{attribute 'GeneratedUsingTerminal: EP1312-0001-0016'}
{attribute addProperty BoxType "EP1312-0001-0016"}
{attribute addProperty Id "A_0038_EP1518_0002_0016EP1518_CC44258859A_0039_EP1518_0002_0017EP1518_CC44258859A_0040_EP1518_0002_0018EP1518_CC44258859A_0041_EP1518_0002_0019EP1518_CC44258859A_0042_EP1809_0021_0016EP1809_32157CFD20A_0043_EP1809_0021_0017EP1809_32157CFD20A_0044_EP1809_0022_0017EP1809_32157CFD20A_0045_EP1809_0022_0018EP1809_32157CFD20A_0046_EP1809_0042_0018EP1809_AA84A50E20A_0047_EP1809_0042_0019EP1809_8E14C81620A_0048_EP1816_0003_0016EP1816_73178B5432A_0049_EP1816_0008_0016EP1816_03D8810930A_0050_EP1816_0008_0017EP1816_03D8810930A_0051_EP1816_0008_0018EP1816_5E50D3DD30A_0052_EP1816_0008_0019EP1816_5E50D3DD30A_0053_EP1816_0008_0020EP1816_5E50D3DD30A_0054_EP1816_1008_0016EP1816_F50297FE32A_0055_EP1816_1008_0017EP1816_F50297FE32A_0056_EP1816_3008_0016EP1816_CABD51E656A_0057_EP1816_3008_0017EP1816_CABD51E656A_0058_EP1816_3008_0018EP1816_CABD51E656A_0059_EP1819_0021_0016EP1819_32157CFD20A_0060_EP1819_0021_0017EP1819_32157CFD20A_0061_EP1819_0022_0016EP1819_32157CFD20A_0062_EP1819_0022_0017EP1819_32157CFD20A_0063_EP1859_0042_0018EP1859_B704EC1A20A_0064_EP1859_0042_0019EP1859_B9D5A78520"}
{attribute addProperty CRC "554975917"}
{attribute addProperty Size "890"}
TYPE A_0037_EP1312_0001_0016_211442AD EXTENDS EP1312_1FC0878B :
STRUCT
	{attribute addProperty Name "A_0038_EP1518_0002_0016"}
	{attribute addProperty PreviousPort "A_0037(EP1312-0001-0016) : D"}
	A_0038_EP1518_0002_0016 : EP1518_CC442588;
	{attribute addProperty Name "A_0039_EP1518_0002_0017"}
	{attribute addProperty PreviousPort "A_0038(EP1518-0002-0016) : B"}
	A_0039_EP1518_0002_0017 : EP1518_CC442588;
	{attribute addProperty Name "A_0040_EP1518_0002_0018"}
	{attribute addProperty PreviousPort "A_0039(EP1518-0002-0017) : B"}
	A_0040_EP1518_0002_0018 : EP1518_CC442588;
	{attribute addProperty Name "A_0041_EP1518_0002_0019"}
	{attribute addProperty PreviousPort "A_0040(EP1518-0002-0018) : B"}
	A_0041_EP1518_0002_0019 : EP1518_CC442588;
	{attribute addProperty Name "A_0042_EP1809_0021_0016"}
	{attribute addProperty PreviousPort "A_0041(EP1518-0002-0019) : B"}
	A_0042_EP1809_0021_0016 : EP1809_32157CFD;
	{attribute addProperty Name "A_0043_EP1809_0021_0017"}
	{attribute addProperty PreviousPort "A_0042(EP1809-0021-0016) : B"}
	A_0043_EP1809_0021_0017 : EP1809_32157CFD;
	{attribute addProperty Name "A_0044_EP1809_0022_0017"}
	{attribute addProperty PreviousPort "A_0043(EP1809-0021-0017) : B"}
	A_0044_EP1809_0022_0017 : EP1809_32157CFD;
	{attribute addProperty Name "A_0045_EP1809_0022_0018"}
	{attribute addProperty PreviousPort "A_0044(EP1809-0022-0017) : B"}
	A_0045_EP1809_0022_0018 : EP1809_32157CFD;
	{attribute addProperty Name "A_0046_EP1809_0042_0018"}
	{attribute addProperty PreviousPort "A_0045(EP1809-0022-0018) : B"}
	A_0046_EP1809_0042_0018 : EP1809_AA84A50E;
	{attribute addProperty Name "A_0047_EP1809_0042_0019"}
	{attribute addProperty PreviousPort "A_0046(EP1809-0042-0018) : B"}
	A_0047_EP1809_0042_0019 : EP1809_8E14C816;
	{attribute addProperty Name "A_0048_EP1816_0003_0016"}
	{attribute addProperty PreviousPort "A_0047(EP1809-0042-0019) : B"}
	A_0048_EP1816_0003_0016 : EP1816_73178B54;
	{attribute addProperty Name "A_0049_EP1816_0008_0016"}
	{attribute addProperty PreviousPort "A_0048(EP1816-0003-0016) : B"}
	A_0049_EP1816_0008_0016 : EP1816_03D88109;
	{attribute addProperty Name "A_0050_EP1816_0008_0017"}
	{attribute addProperty PreviousPort "A_0049(EP1816-0008-0016) : B"}
	A_0050_EP1816_0008_0017 : EP1816_03D88109;
	{attribute addProperty Name "A_0051_EP1816_0008_0018"}
	{attribute addProperty PreviousPort "A_0050(EP1816-0008-0017) : B"}
	A_0051_EP1816_0008_0018 : EP1816_5E50D3DD;
	{attribute addProperty Name "A_0052_EP1816_0008_0019"}
	{attribute addProperty PreviousPort "A_0051(EP1816-0008-0018) : B"}
	A_0052_EP1816_0008_0019 : EP1816_5E50D3DD;
	{attribute addProperty Name "A_0053_EP1816_0008_0020"}
	{attribute addProperty PreviousPort "A_0052(EP1816-0008-0019) : B"}
	A_0053_EP1816_0008_0020 : EP1816_5E50D3DD;
	{attribute addProperty Name "A_0054_EP1816_1008_0016"}
	{attribute addProperty PreviousPort "A_0053(EP1816-0008-0020) : B"}
	A_0054_EP1816_1008_0016 : EP1816_F50297FE;
	{attribute addProperty Name "A_0055_EP1816_1008_0017"}
	{attribute addProperty PreviousPort "A_0054(EP1816-1008-0016) : B"}
	A_0055_EP1816_1008_0017 : EP1816_F50297FE;
	{attribute addProperty Name "A_0056_EP1816_3008_0016"}
	{attribute addProperty PreviousPort "A_0055(EP1816-1008-0017) : B"}
	A_0056_EP1816_3008_0016 : EP1816_CABD51E6;
	{attribute addProperty Name "A_0057_EP1816_3008_0017"}
	{attribute addProperty PreviousPort "A_0056(EP1816-3008-0016) : B"}
	A_0057_EP1816_3008_0017 : EP1816_CABD51E6;
	{attribute addProperty Name "A_0058_EP1816_3008_0018"}
	{attribute addProperty PreviousPort "A_0057(EP1816-3008-0017) : B"}
	A_0058_EP1816_3008_0018 : EP1816_CABD51E6;
	{attribute addProperty Name "A_0059_EP1819_0021_0016"}
	{attribute addProperty PreviousPort "A_0058(EP1816-3008-0018) : B"}
	A_0059_EP1819_0021_0016 : EP1819_32157CFD;
	{attribute addProperty Name "A_0060_EP1819_0021_0017"}
	{attribute addProperty PreviousPort "A_0059(EP1819-0021-0016) : B"}
	A_0060_EP1819_0021_0017 : EP1819_32157CFD;
	{attribute addProperty Name "A_0061_EP1819_0022_0016"}
	{attribute addProperty PreviousPort "A_0060(EP1819-0021-0017) : B"}
	A_0061_EP1819_0022_0016 : EP1819_32157CFD;
	{attribute addProperty Name "A_0062_EP1819_0022_0017"}
	{attribute addProperty PreviousPort "A_0061(EP1819-0022-0016) : B"}
	A_0062_EP1819_0022_0017 : EP1819_32157CFD;
	{attribute addProperty Name "A_0063_EP1859_0042_0018"}
	{attribute addProperty PreviousPort "A_0062(EP1819-0022-0017) : B"}
	A_0063_EP1859_0042_0018 : EP1859_B704EC1A;
	{attribute addProperty Name "A_0064_EP1859_0042_0019"}
	{attribute addProperty PreviousPort "A_0063(EP1859-0042-0018) : B"}
	A_0064_EP1859_0042_0019 : EP1859_B9D5A785;
END_STRUCT
END_TYPE

(* stored: Version 1.2.0.0, ProductVersion 3.1.4024.9
   DUT A_0037_EP1312_0001_0016_211442AD: Id {e0bec23f-b433-4ee7-86f5-85c4ff9f79c8} *)
